SUBAPPLICATION Uebung_081 (* Beispiel für E_CTD *)
  (* Standard: 61499-2; Description: Beispiel für E_CTD Aufwärts zählen UAO Curriculum Module 3 - The IEC 61499 Standard, Seite 93 *)
  (* Version 1.0, 2023-10-23, franz *)
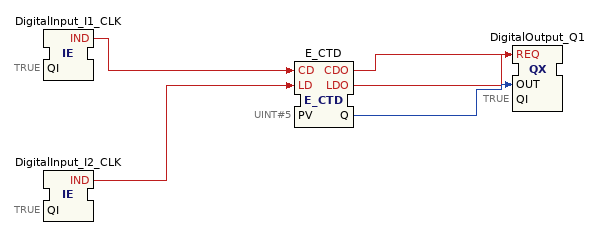
  FBS
    DigitalOutput_Q1 : QX(QI := TRUE);
    DigitalInput_I1_CLK : IE(QI := TRUE);
    E_CTD : E_CTD(PV := UINT#5);
    DigitalInput_I2_CLK : IE(QI := TRUE);
  END_FBS
  EVENT_CONNECTIONS
    DigitalInput_I1_CLK.IND TO E_CTD.CD;
    E_CTD.CDO TO DigitalOutput_Q1.REQ;
    E_CTD.LDO TO DigitalOutput_Q1.REQ;
    DigitalInput_I2_CLK.IND TO E_CTD.LD;
  END_CONNECTIONS
  DATA_CONNECTIONS
    E_CTD.Q TO DigitalOutput_Q1.OUT;
  END_CONNECTIONS
END_SUBAPPLICATION
